// Mitsubishi GX Works2 project: shrimp_load_v01   PLC: FX3G
// Carga de PLC para monitoreo de piscina de camarones

PROGRAM MAIN
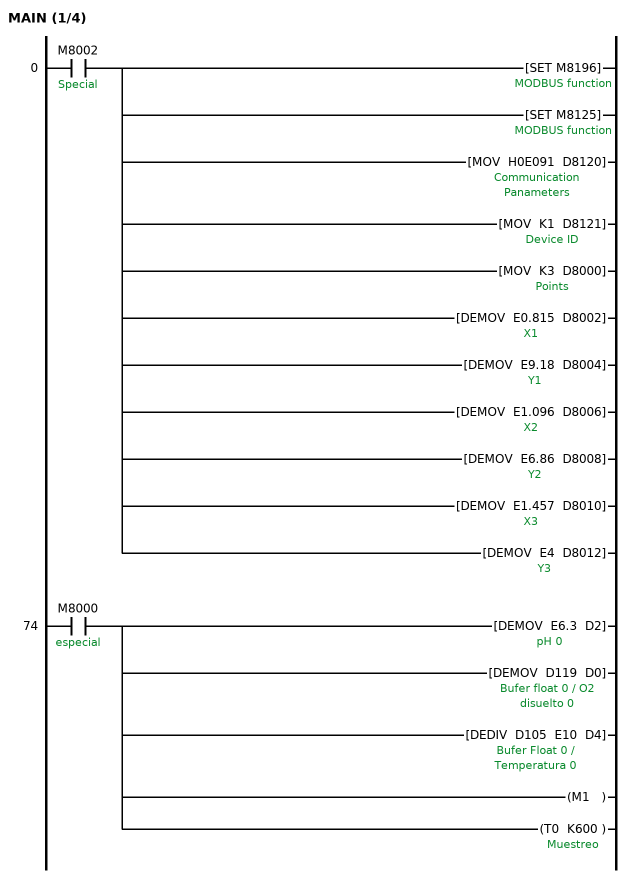
0     LD      M8002  ; Special
      SET     M8196  ; MODBUS function
      SET     M8125  ; MODBUS function
      MOV     H0E091 D8120  ; Communication Panameters
      MOV     K1 D8121  ; Device ID
      MOV     K3 D8000  ; Points
      DEMOV   E0.815 D8002  ; X1
      DEMOV   E9.18 D8004  ; Y1
      DEMOV   E1.096 D8006  ; X2
      DEMOV   E6.86 D8008  ; Y2
      DEMOV   E1.457 D8010  ; X3
      DEMOV   E4 D8012  ; Y3
74    LD      M8000  ; especial
      DEMOV   E6.3 D2  ; pH 0
      DEMOV   D119 D0  ; Bufer float 0 / O2 disuelto 0
      DEDIV   D105 E10 D4  ; Bufer Float 0 / Temperatura 0
      OUT     M1
      OUT     T0 K600  ; Muestreo
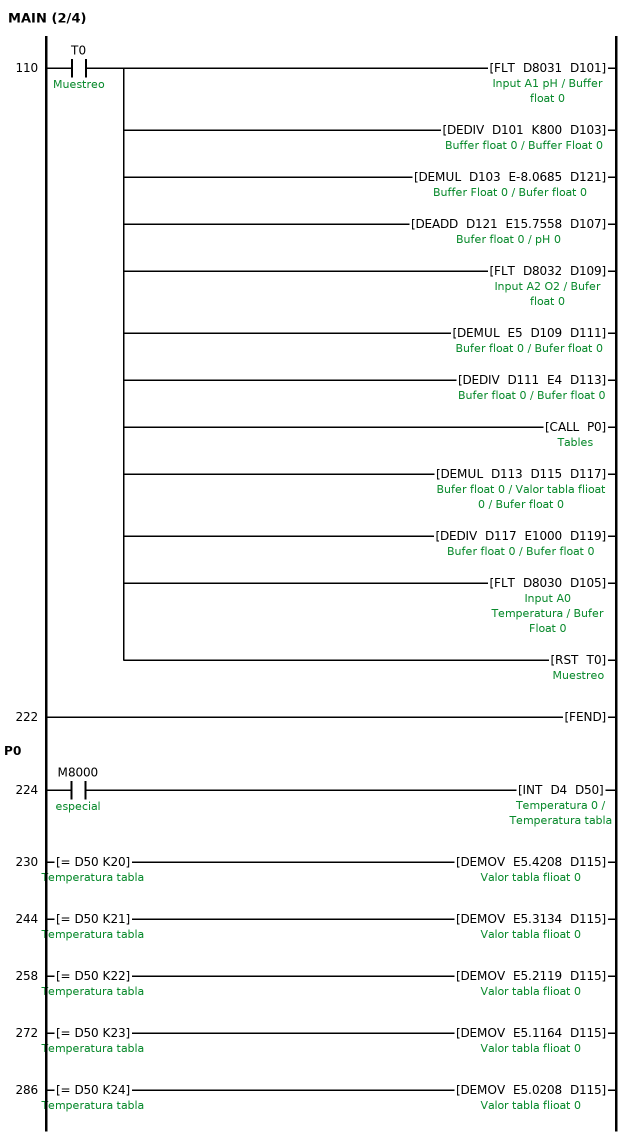
110   LD      T0  ; Muestreo
      FLT     D8031 D101  ; Input A1 pH / Buffer float 0
      DEDIV   D101 K800 D103  ; Buffer Float 0
      DEMUL   D103 E-8.0685 D121  ; Bufer float 0
      DEADD   D121 E15.7558 D107  ; pH 0
      FLT     D8032 D109  ; Input A2 O2 / Bufer float 0
      DEMUL   E5 D109 D111  ; Bufer float 0
      DEDIV   D111 E4 D113  ; Bufer float 0
      CALL    P0  ; Tables
      DEMUL   D113 D115 D117  ; Valor tabla flioat 0 / Bufer float 0
      DEDIV   D117 E1000 D119
      FLT     D8030 D105  ; Input A0 Temperatura
      RST     T0  ; Muestreo
222   FEND
      P0
224   LD      M8000  ; especial
      INT     D4 D50  ; Temperatura tabla
230   LD=     D50 K20  ; Temperatura tabla
      DEMOV   E5.4208 D115
244   LD=     D50 K21  ; Temperatura tabla
      DEMOV   E5.3134 D115
258   LD=     D50 K22  ; Temperatura tabla
      DEMOV   E5.2119 D115
272   LD=     D50 K23  ; Temperatura tabla
      DEMOV   E5.1164 D115
286   LD=     D50 K24  ; Temperatura tabla
      DEMOV   E5.0208 D115
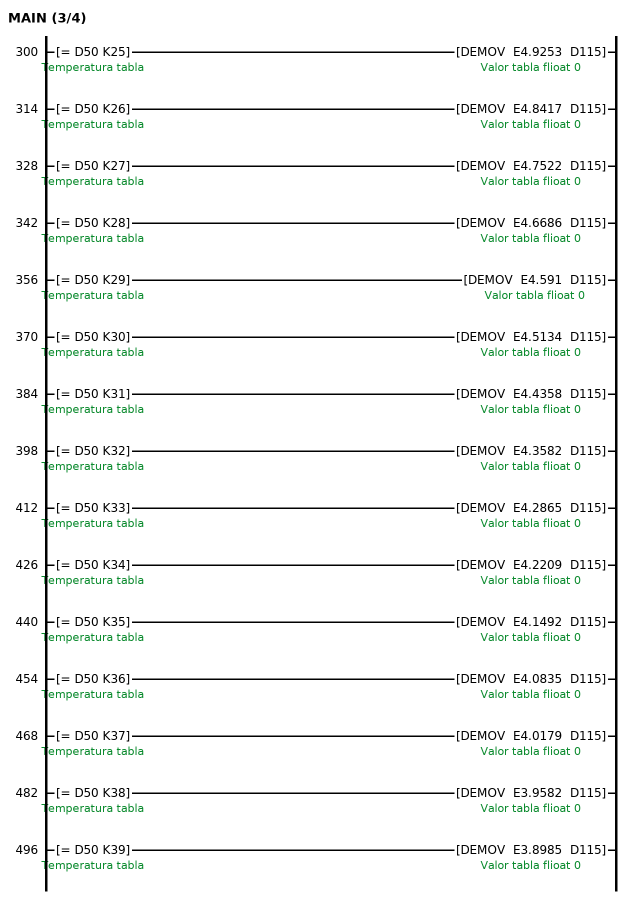
300   LD=     D50 K25  ; Temperatura tabla
      DEMOV   E4.9253 D115
314   LD=     D50 K26  ; Temperatura tabla
      DEMOV   E4.8417 D115
328   LD=     D50 K27  ; Temperatura tabla
      DEMOV   E4.7522 D115
342   LD=     D50 K28  ; Temperatura tabla
      DEMOV   E4.6686 D115
356   LD=     D50 K29  ; Temperatura tabla
      DEMOV   E4.591 D115
370   LD=     D50 K30  ; Temperatura tabla
      DEMOV   E4.5134 D115
384   LD=     D50 K31  ; Temperatura tabla
      DEMOV   E4.4358 D115
398   LD=     D50 K32  ; Temperatura tabla
      DEMOV   E4.3582 D115
412   LD=     D50 K33  ; Temperatura tabla
      DEMOV   E4.2865 D115
426   LD=     D50 K34  ; Temperatura tabla
      DEMOV   E4.2209 D115
440   LD=     D50 K35  ; Temperatura tabla
      DEMOV   E4.1492 D115
454   LD=     D50 K36  ; Temperatura tabla
      DEMOV   E4.0835 D115
468   LD=     D50 K37  ; Temperatura tabla
      DEMOV   E4.0179 D115
482   LD=     D50 K38  ; Temperatura tabla
      DEMOV   E3.9582 D115
496   LD=     D50 K39  ; Temperatura tabla
      DEMOV   E3.8985 D115
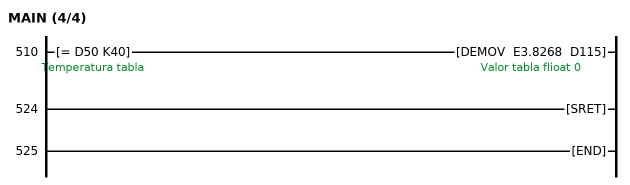
510   LD=     D50 K40  ; Temperatura tabla
      DEMOV   E3.8268 D115
524   SRET
525   END
END_PROGRAM

// device comments not shown above
D1  ; O2 disuelto 1
D3  ; pH 1
D5  ; Temperatura 1
D100  ; Buffer
D102  ; Buffer Float 1
D104  ; Bufer Float 1
D108  ; pH 1
D110  ; Bufer FLoat 1
D200  ; Buffer Float
D204  ; Bufer float
T200  ; Muestra
